{attribute 'qualified_only'}
TYPE ENUM_WFS_States :
(
    Unknown := 0,
    OUT := 1,
    TARGET1 := 2,
    TARGET2 := 3,
    TARGET3 := 4,
    TARGET4 := 5,
    TARGET5 := 6
);
END_TYPE

(* stored: Version 1.1.0.1
   DUT ENUM_WFS_States: Id {3453a453-2671-4525-8745-914037e14ff2} *)
